(* Logix 5000 project; controller SX_V040001_C001 vendor 1 type 14 code 77 rev 16.22; software revision 16.04; part 7 of 35 *)
(* tags used below, declared in another part *)
   ALARM_BITS : INT[10];
   ALL_KINDS : INT[90];
   average_current : DINT;
   DRIVE : INT[32];
   DRIVE_INTERVAL : INT[8];
   EMPTYING : INT[18];
   FP_ALARM_EXIST : BOOL;
   G_AInput : DINT[8];
   G_DInput : DINT[3];
   G_DOutput : DINT[3];
   loading : INT[19];
   m_alarm_exist : BOOL;
   m_alarm_horn : BOOL;
   m_notstop : BOOL;
   METERING : INT[44];
   PARAMETER : INT[501];
   pointer_dump_current : DINT;
   RECIPE_GENERAL : INT[405];
   T_MET12_END : TIMER;
   T_MET13_END : TIMER;
   T_MET14_END : TIMER;
   T_MET_VALVE_13 : TIMER;
   T_MET_VALVE_14 : TIMER;
   TEMP : INT[14];
(* MainProgram, continued *)

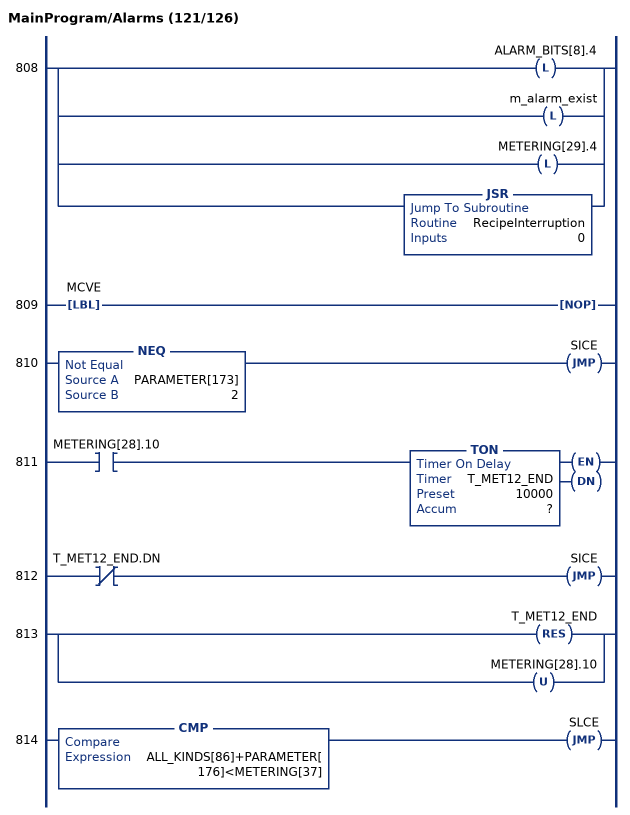
   [picture p142: MainProgram/Alarms rungs 808-814]
   808: [OTL(ALARM_BITS[8].4) ,OTL(m_alarm_exist) ,OTL(METERING[29].4) ,JSR(RecipeInterruption,0) ];
   809: LBL(MCVE)NOP();
   810: NEQ(PARAMETER[173],2)JMP(SICE);
   811: XIC(METERING[28].10)TON(T_MET12_END,?,?);
   812: XIO(T_MET12_END.DN)JMP(SICE);
   813: [RES(T_MET12_END) ,OTU(METERING[28].10) ];
   814: CMP(ALL_KINDS[86]+PARAMETER[176]<METERING[37])JMP(SLCE);
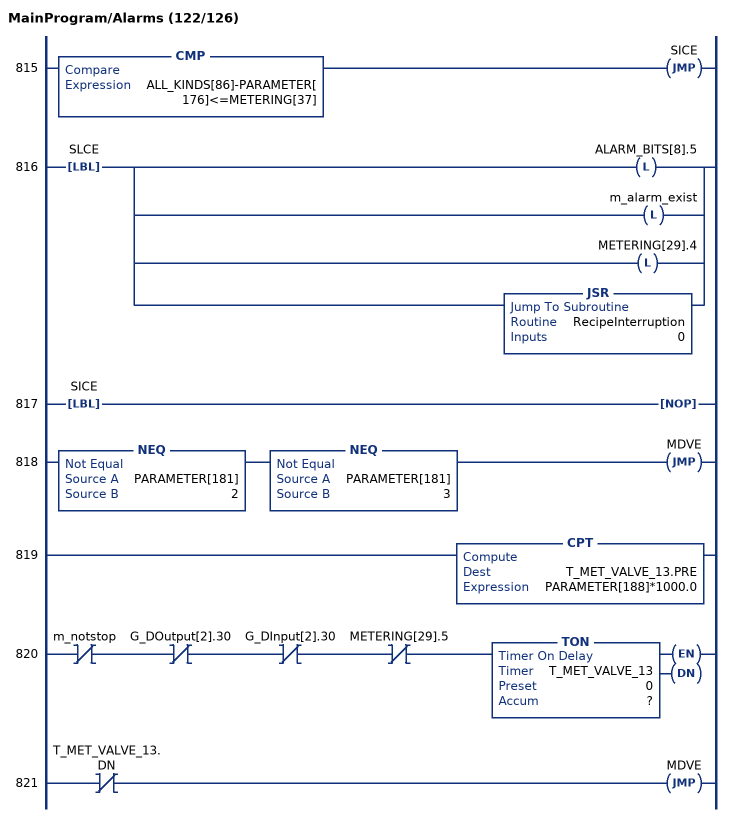
   815: CMP(ALL_KINDS[86]-PARAMETER[176]<=METERING[37])JMP(SICE);
   816: LBL(SLCE)[OTL(ALARM_BITS[8].5) ,OTL(m_alarm_exist) ,OTL(METERING[29].4) ,JSR(RecipeInterruption,0) ];
   817: LBL(SICE)NOP();
   818: NEQ(PARAMETER[181],2)NEQ(PARAMETER[181],3)JMP(MDVE);
   819: CPT(T_MET_VALVE_13.PRE,PARAMETER[188]*1000.0);
   820: XIO(m_notstop)XIO(G_DOutput[2].30)XIO(G_DInput[2].30)XIO(METERING[29].5)TON(T_MET_VALVE_13,?,?);
   821: XIO(T_MET_VALVE_13.DN)JMP(MDVE);
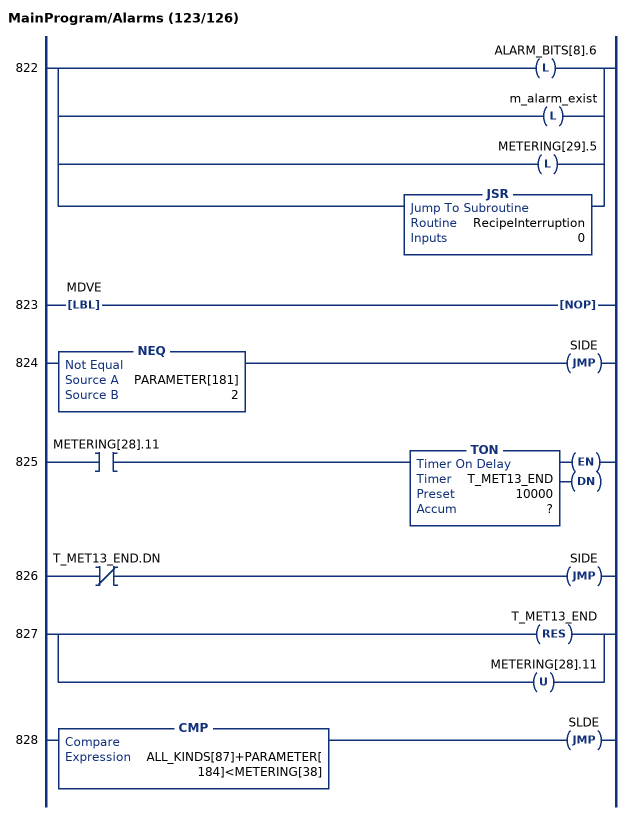
   822: [OTL(ALARM_BITS[8].6) ,OTL(m_alarm_exist) ,OTL(METERING[29].5) ,JSR(RecipeInterruption,0) ];
   823: LBL(MDVE)NOP();
   824: NEQ(PARAMETER[181],2)JMP(SIDE);
   825: XIC(METERING[28].11)TON(T_MET13_END,?,?);
   826: XIO(T_MET13_END.DN)JMP(SIDE);
   827: [RES(T_MET13_END) ,OTU(METERING[28].11) ];
   828: CMP(ALL_KINDS[87]+PARAMETER[184]<METERING[38])JMP(SLDE);
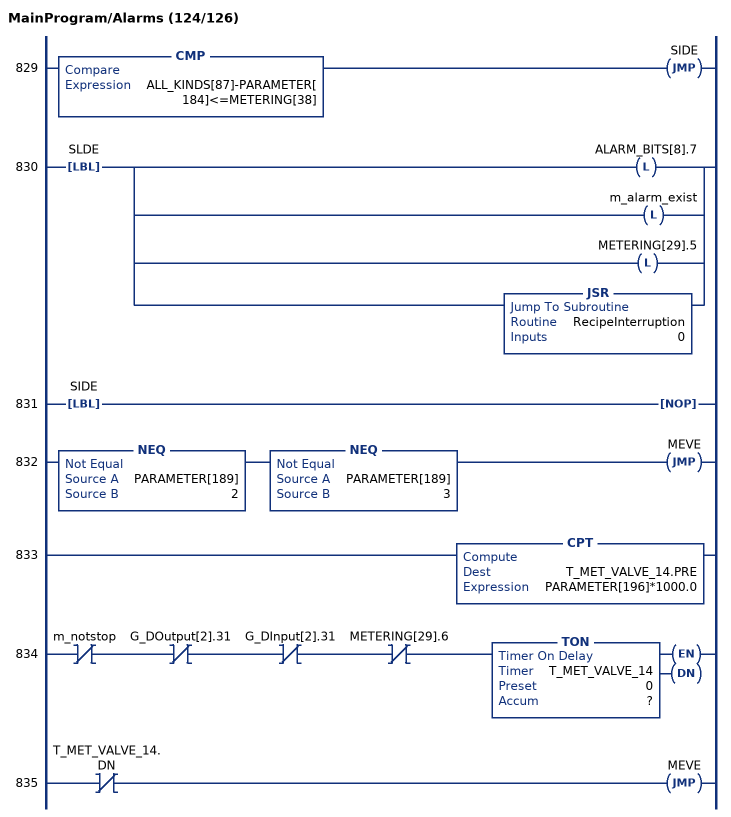
   829: CMP(ALL_KINDS[87]-PARAMETER[184]<=METERING[38])JMP(SIDE);
   830: LBL(SLDE)[OTL(ALARM_BITS[8].7) ,OTL(m_alarm_exist) ,OTL(METERING[29].5) ,JSR(RecipeInterruption,0) ];
   831: LBL(SIDE)NOP();
   832: NEQ(PARAMETER[189],2)NEQ(PARAMETER[189],3)JMP(MEVE);
   833: CPT(T_MET_VALVE_14.PRE,PARAMETER[196]*1000.0);
   834: XIO(m_notstop)XIO(G_DOutput[2].31)XIO(G_DInput[2].31)XIO(METERING[29].6)TON(T_MET_VALVE_14,?,?);
   835: XIO(T_MET_VALVE_14.DN)JMP(MEVE);
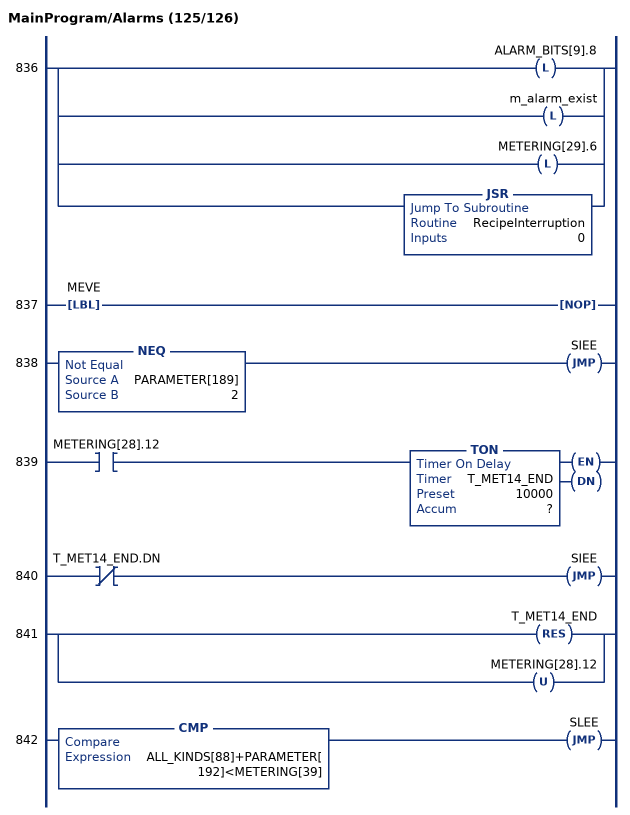
   836: [OTL(ALARM_BITS[9].8) ,OTL(m_alarm_exist) ,OTL(METERING[29].6) ,JSR(RecipeInterruption,0) ];
   837: LBL(MEVE)NOP();
   838: NEQ(PARAMETER[189],2)JMP(SIEE);
   839: XIC(METERING[28].12)TON(T_MET14_END,?,?);
   840: XIO(T_MET14_END.DN)JMP(SIEE);
   841: [RES(T_MET14_END) ,OTU(METERING[28].12) ];
   842: CMP(ALL_KINDS[88]+PARAMETER[192]<METERING[39])JMP(SLEE);
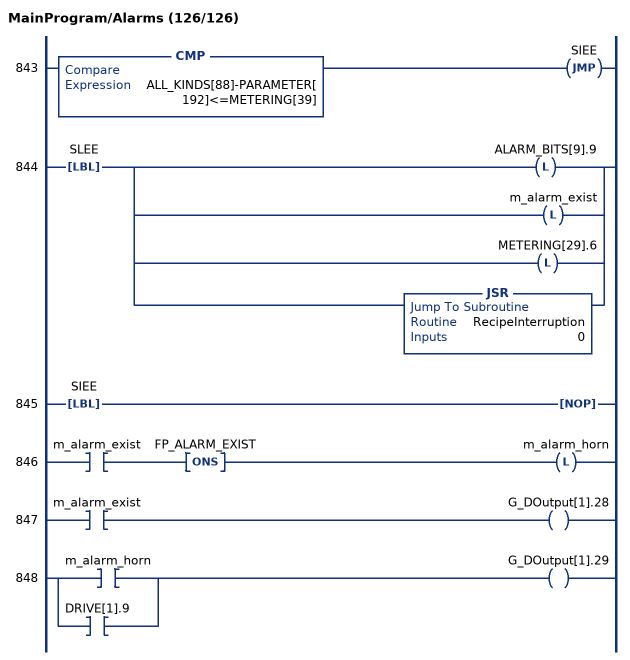
   843: CMP(ALL_KINDS[88]-PARAMETER[192]<=METERING[39])JMP(SIEE);
   844: LBL(SLEE)[OTL(ALARM_BITS[9].9) ,OTL(m_alarm_exist) ,OTL(METERING[29].6) ,JSR(RecipeInterruption,0) ];
   845: LBL(SIEE)NOP();
   846: XIC(m_alarm_exist)ONS(FP_ALARM_EXIST)OTL(m_alarm_horn);
   847: XIC(m_alarm_exist)OTE(G_DOutput[1].28);
   848: [XIC(m_alarm_horn) ,XIC(DRIVE[1].9) ]OTE(G_DOutput[1].29);
END_ROUTINE

ROUTINE AnalogInput   (* ladder *)
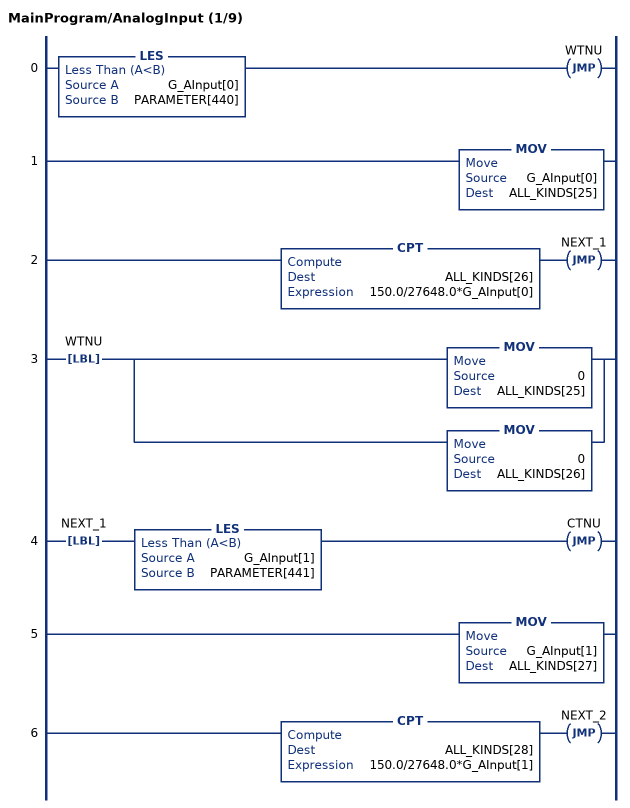
   0: LES(G_AInput[0],PARAMETER[440])JMP(WTNU);
   1: MOV(G_AInput[0],ALL_KINDS[25]);
   2: CPT(ALL_KINDS[26],150.0/27648.0*G_AInput[0])JMP(NEXT_1);
   3: LBL(WTNU)[MOV(0,ALL_KINDS[25]) ,MOV(0,ALL_KINDS[26]) ];
   4: LBL(NEXT_1)LES(G_AInput[1],PARAMETER[441])JMP(CTNU);
   5: MOV(G_AInput[1],ALL_KINDS[27]);
   6: CPT(ALL_KINDS[28],150.0/27648.0*G_AInput[1])JMP(NEXT_2);
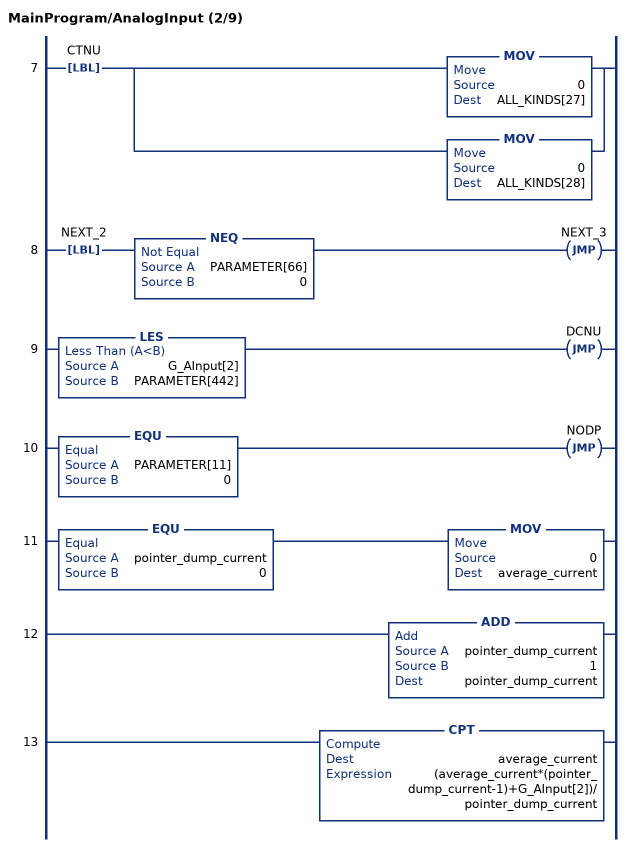
   7: LBL(CTNU)[MOV(0,ALL_KINDS[27]) ,MOV(0,ALL_KINDS[28]) ];
   8: LBL(NEXT_2)NEQ(PARAMETER[66],0)JMP(NEXT_3);
   9: LES(G_AInput[2],PARAMETER[442])JMP(DCNU);
   10: EQU(PARAMETER[11],0)JMP(NODP);
   11: EQU(pointer_dump_current,0)MOV(0,average_current);
   12: ADD(pointer_dump_current,1,pointer_dump_current);
   13: CPT(average_current,(average_current*(pointer_dump_current-1)+G_AInput[2])/pointer_dump_current);
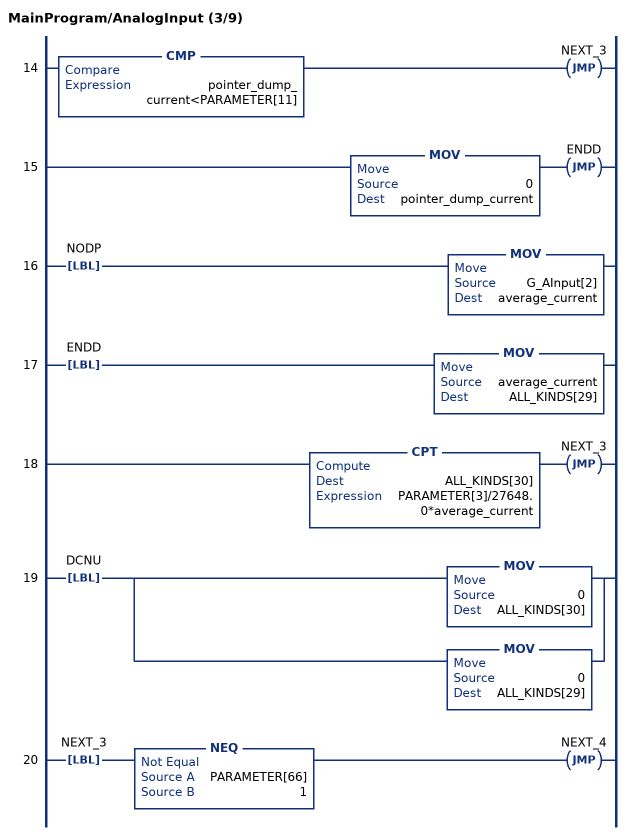
   14: CMP(pointer_dump_current<PARAMETER[11])JMP(NEXT_3);
   15: MOV(0,pointer_dump_current)JMP(ENDD);
   16: LBL(NODP)MOV(G_AInput[2],average_current);
   17: LBL(ENDD)MOV(average_current,ALL_KINDS[29]);
   18: CPT(ALL_KINDS[30],PARAMETER[3]/27648.0*average_current)JMP(NEXT_3);
   19: LBL(DCNU)[MOV(0,ALL_KINDS[30]) ,MOV(0,ALL_KINDS[29]) ];
   20: LBL(NEXT_3)NEQ(PARAMETER[66],1)JMP(NEXT_4);
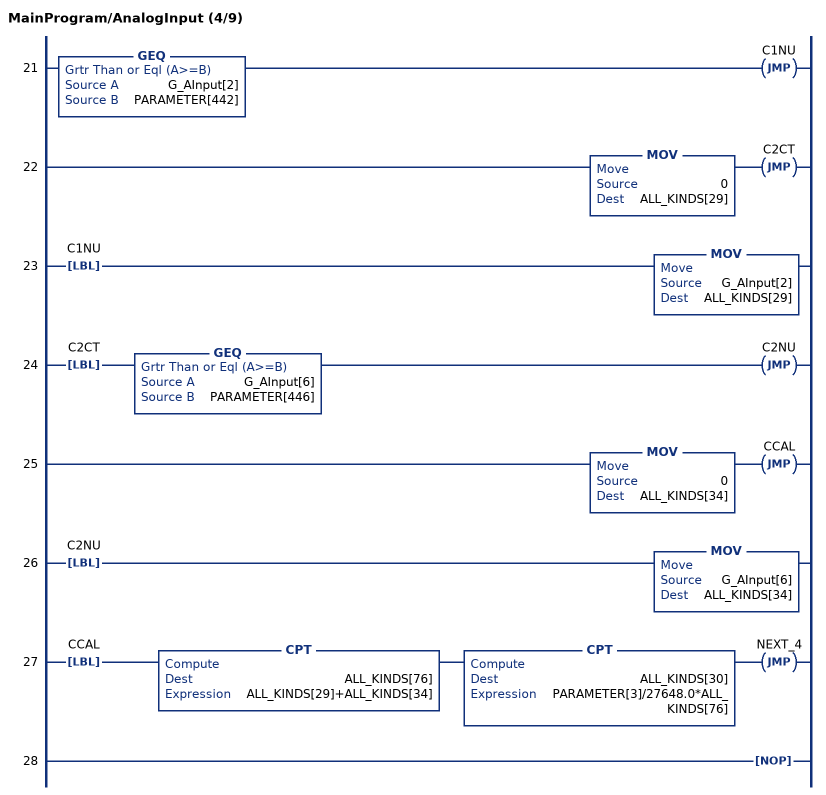
   21: GEQ(G_AInput[2],PARAMETER[442])JMP(C1NU);
   22: MOV(0,ALL_KINDS[29])JMP(C2CT);
   23: LBL(C1NU)MOV(G_AInput[2],ALL_KINDS[29]);
   24: LBL(C2CT)GEQ(G_AInput[6],PARAMETER[446])JMP(C2NU);
   25: MOV(0,ALL_KINDS[34])JMP(CCAL);
   26: LBL(C2NU)MOV(G_AInput[6],ALL_KINDS[34]);
   27: LBL(CCAL)CPT(ALL_KINDS[76],ALL_KINDS[29]+ALL_KINDS[34])CPT(ALL_KINDS[30],PARAMETER[3]/27648.0*ALL_KINDS[76])JMP(NEXT_4);
   28: NOP();
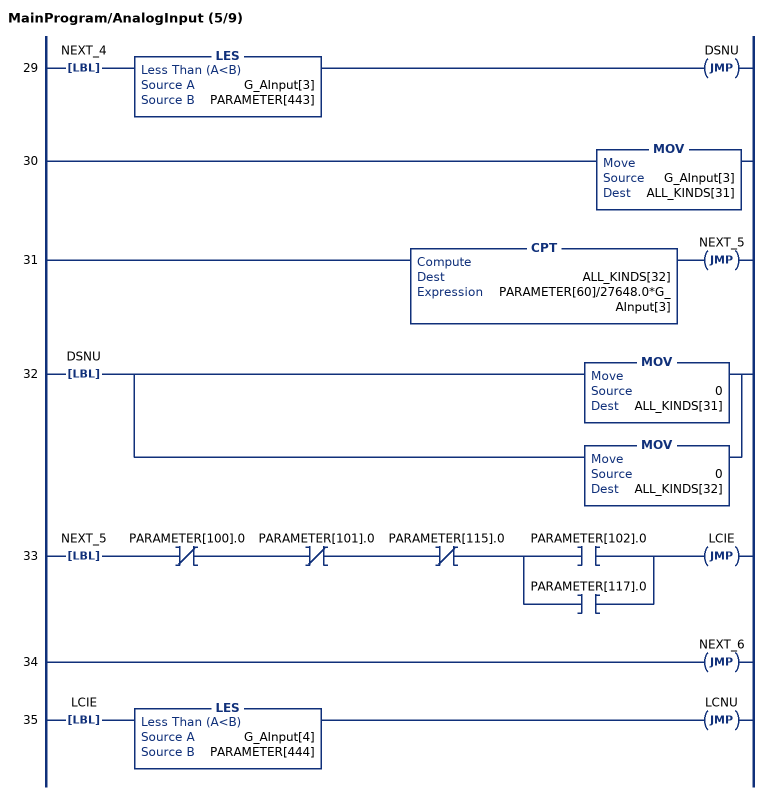
   29: LBL(NEXT_4)LES(G_AInput[3],PARAMETER[443])JMP(DSNU);
   30: MOV(G_AInput[3],ALL_KINDS[31]);
   31: CPT(ALL_KINDS[32],PARAMETER[60]/27648.0*G_AInput[3])JMP(NEXT_5);
   32: LBL(DSNU)[MOV(0,ALL_KINDS[31]) ,MOV(0,ALL_KINDS[32]) ];
   33: LBL(NEXT_5)XIO(PARAMETER[100].0)XIO(PARAMETER[101].0)XIO(PARAMETER[115].0)[XIC(PARAMETER[102].0) ,XIC(PARAMETER[117].0) ]JMP(LCIE);
   34: JMP(NEXT_6);
   35: LBL(LCIE)LES(G_AInput[4],PARAMETER[444])JMP(LCNU);
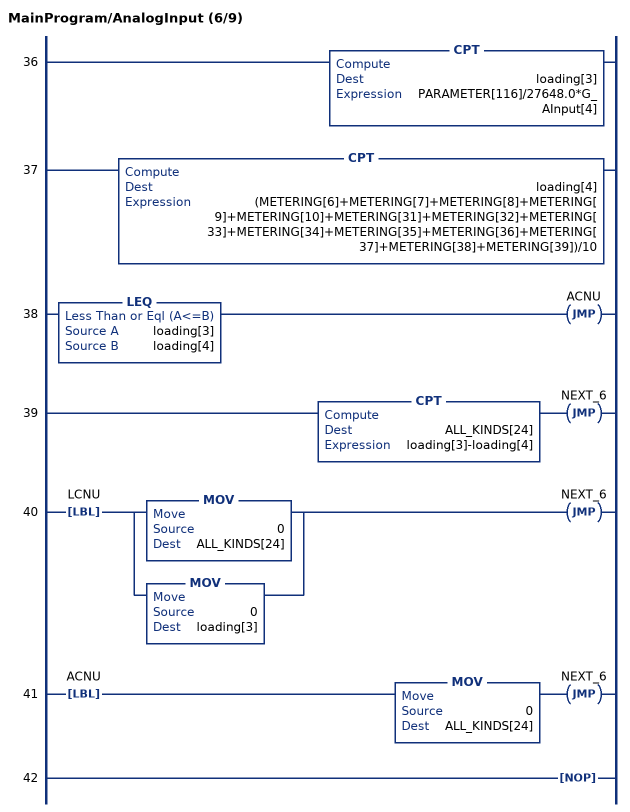
   36: CPT(loading[3],PARAMETER[116]/27648.0*G_AInput[4]);
   37: CPT(loading[4],(METERING[6]+METERING[7]+METERING[8]+METERING[9]+METERING[10]+METERING[31]+METERING[32]+METERING[33]+METERING[34]+METERING[35]+METERING[36]+METERING[37]+METERING[38]+METERING[39])/10);
   38: LEQ(loading[3],loading[4])JMP(ACNU);
   39: CPT(ALL_KINDS[24],loading[3]-loading[4])JMP(NEXT_6);
   40: LBL(LCNU)[MOV(0,ALL_KINDS[24]) ,MOV(0,loading[3]) ]JMP(NEXT_6);
   41: LBL(ACNU)MOV(0,ALL_KINDS[24])JMP(NEXT_6);
   42: NOP();
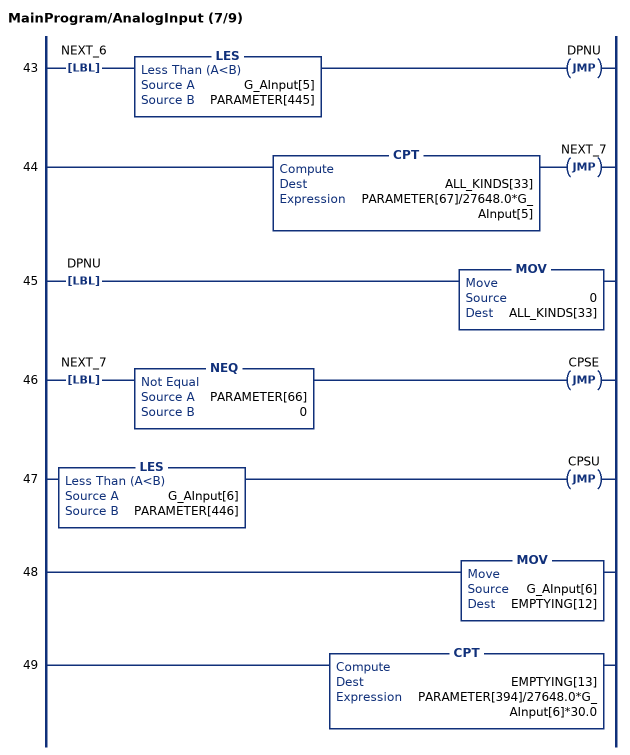
   43: LBL(NEXT_6)LES(G_AInput[5],PARAMETER[445])JMP(DPNU);
   44: CPT(ALL_KINDS[33],PARAMETER[67]/27648.0*G_AInput[5])JMP(NEXT_7);
   45: LBL(DPNU)MOV(0,ALL_KINDS[33]);
   46: LBL(NEXT_7)NEQ(PARAMETER[66],0)JMP(CPSE);
   47: LES(G_AInput[6],PARAMETER[446])JMP(CPSU);
   48: MOV(G_AInput[6],EMPTYING[12]);
   49: CPT(EMPTYING[13],PARAMETER[394]/27648.0*G_AInput[6]*30.0);
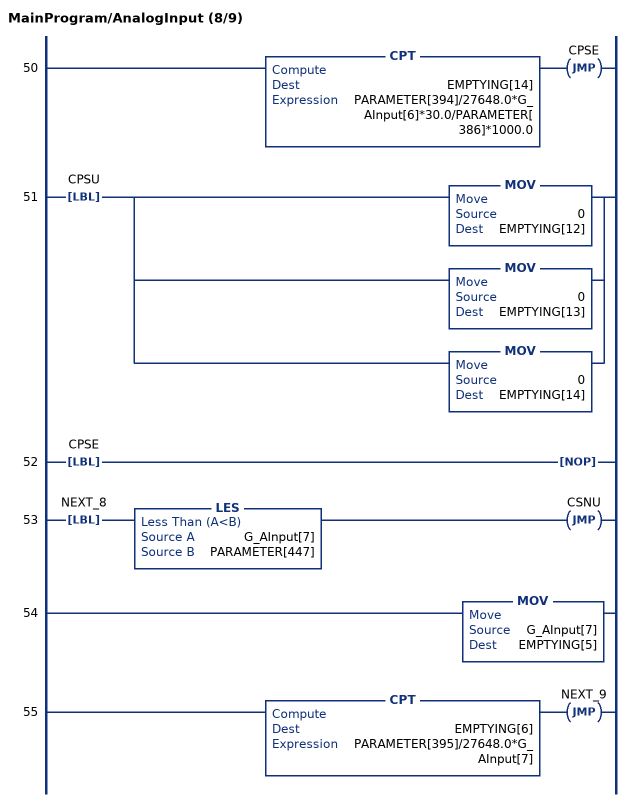
   50: CPT(EMPTYING[14],PARAMETER[394]/27648.0*G_AInput[6]*30.0/PARAMETER[386]*1000.0)JMP(CPSE);
   51: LBL(CPSU)[MOV(0,EMPTYING[12]) ,MOV(0,EMPTYING[13]) ,MOV(0,EMPTYING[14]) ];
   52: LBL(CPSE)NOP();
   53: LBL(NEXT_8)LES(G_AInput[7],PARAMETER[447])JMP(CSNU);
   54: MOV(G_AInput[7],EMPTYING[5]);
   55: CPT(EMPTYING[6],PARAMETER[395]/27648.0*G_AInput[7])JMP(NEXT_9);
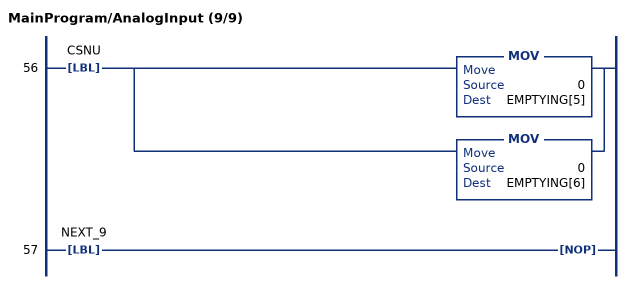
   56: LBL(CSNU)[MOV(0,EMPTYING[5]) ,MOV(0,EMPTYING[6]) ];
   57: LBL(NEXT_9)NOP();
END_ROUTINE

ROUTINE AnalyseRecipe   (* ladder *)
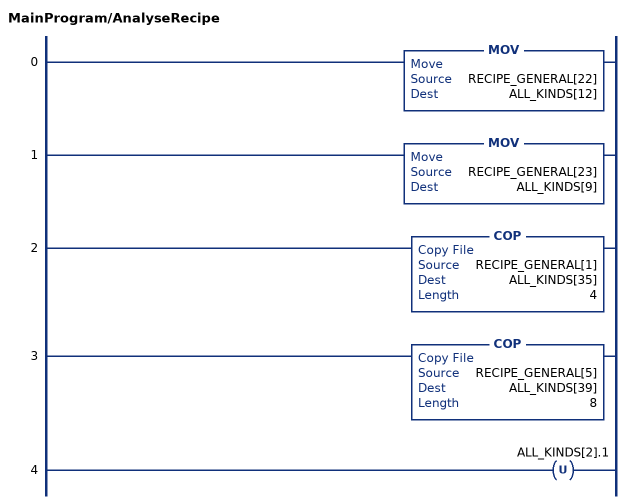
   0: MOV(RECIPE_GENERAL[22],ALL_KINDS[12]);
   1: MOV(RECIPE_GENERAL[23],ALL_KINDS[9]);
   2: COP(RECIPE_GENERAL[1],ALL_KINDS[35],4);
   3: COP(RECIPE_GENERAL[5],ALL_KINDS[39],8);
   4: OTU(ALL_KINDS[2].1);
END_ROUTINE

ROUTINE AnalyseRestart   (* ladder *)
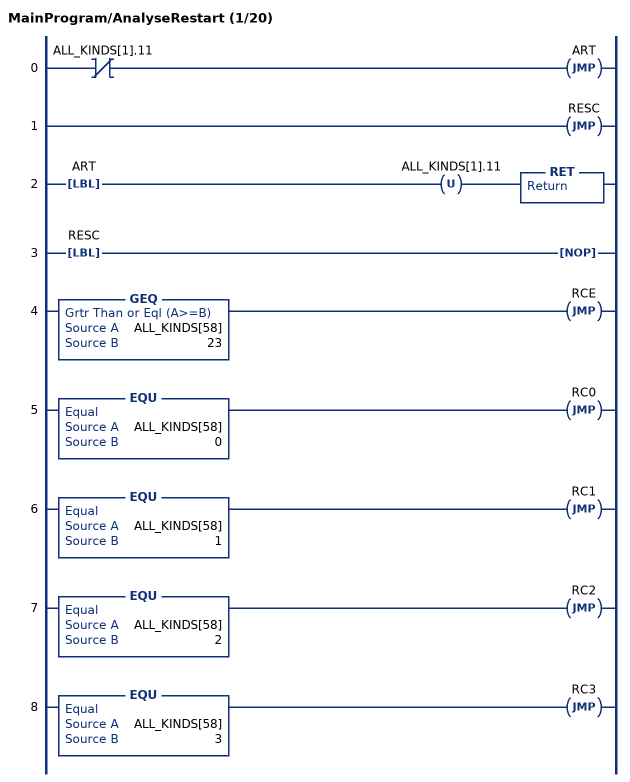
   0: XIO(ALL_KINDS[1].11)JMP(ART);
   1: JMP(RESC);
   2: LBL(ART)OTU(ALL_KINDS[1].11)RET();
   3: LBL(RESC)NOP();
   4: GEQ(ALL_KINDS[58],23)JMP(RCE);
   5: EQU(ALL_KINDS[58],0)JMP(RC0);
   6: EQU(ALL_KINDS[58],1)JMP(RC1);
   7: EQU(ALL_KINDS[58],2)JMP(RC2);
   8: EQU(ALL_KINDS[58],3)JMP(RC3);
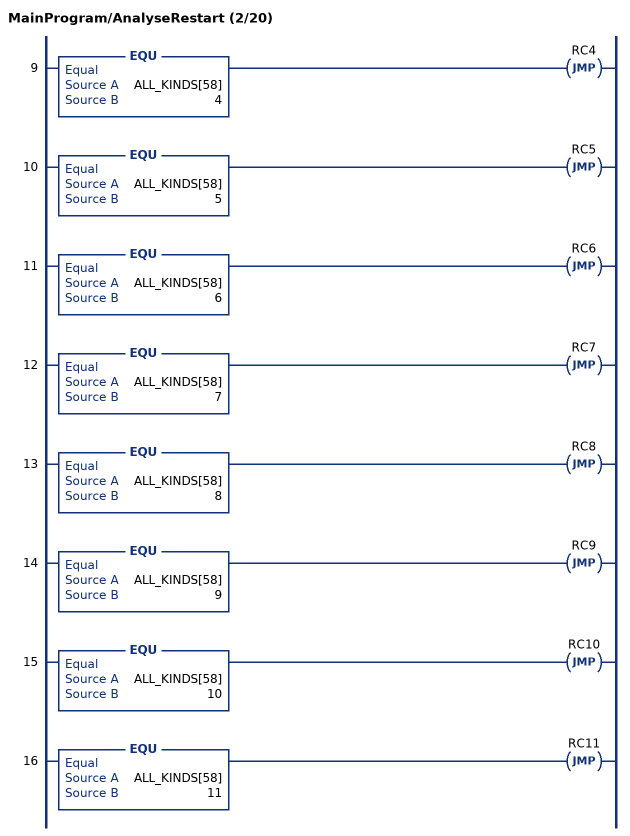
   9: EQU(ALL_KINDS[58],4)JMP(RC4);
   10: EQU(ALL_KINDS[58],5)JMP(RC5);
   11: EQU(ALL_KINDS[58],6)JMP(RC6);
   12: EQU(ALL_KINDS[58],7)JMP(RC7);
   13: EQU(ALL_KINDS[58],8)JMP(RC8);
   14: EQU(ALL_KINDS[58],9)JMP(RC9);
   15: EQU(ALL_KINDS[58],10)JMP(RC10);
   16: EQU(ALL_KINDS[58],11)JMP(RC11);
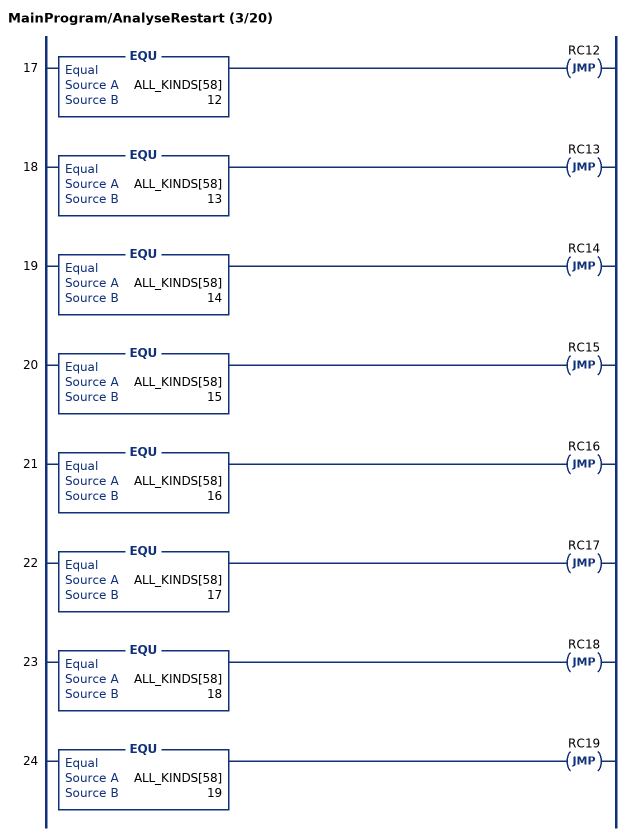
   17: EQU(ALL_KINDS[58],12)JMP(RC12);
   18: EQU(ALL_KINDS[58],13)JMP(RC13);
   19: EQU(ALL_KINDS[58],14)JMP(RC14);
   20: EQU(ALL_KINDS[58],15)JMP(RC15);
   21: EQU(ALL_KINDS[58],16)JMP(RC16);
   22: EQU(ALL_KINDS[58],17)JMP(RC17);
   23: EQU(ALL_KINDS[58],18)JMP(RC18);
   24: EQU(ALL_KINDS[58],19)JMP(RC19);
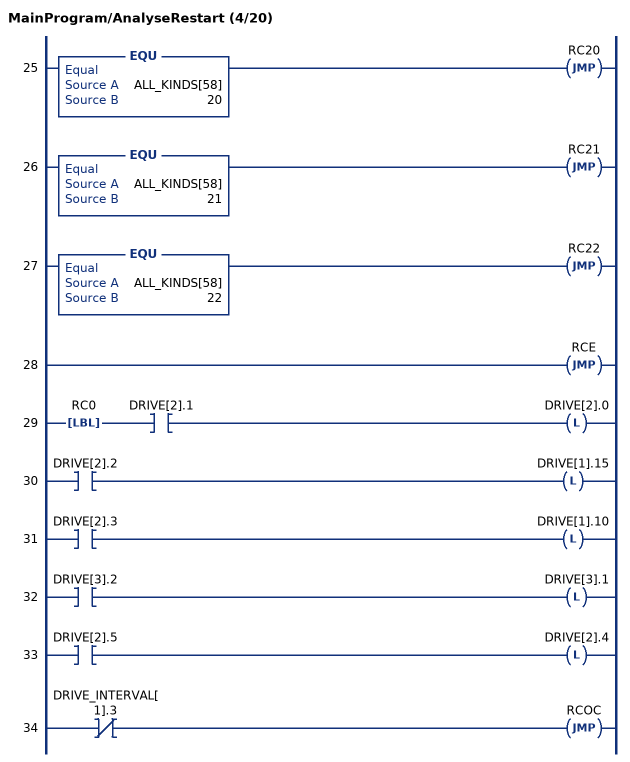
   25: EQU(ALL_KINDS[58],20)JMP(RC20);
   26: EQU(ALL_KINDS[58],21)JMP(RC21);
   27: EQU(ALL_KINDS[58],22)JMP(RC22);
   28: JMP(RCE);
   29: LBL(RC0)XIC(DRIVE[2].1)OTL(DRIVE[2].0);
   30: XIC(DRIVE[2].2)OTL(DRIVE[1].15);
   31: XIC(DRIVE[2].3)OTL(DRIVE[1].10);
   32: XIC(DRIVE[3].2)OTL(DRIVE[3].1);
   33: XIC(DRIVE[2].5)OTL(DRIVE[2].4);
   34: XIO(DRIVE_INTERVAL[1].3)JMP(RCOC);
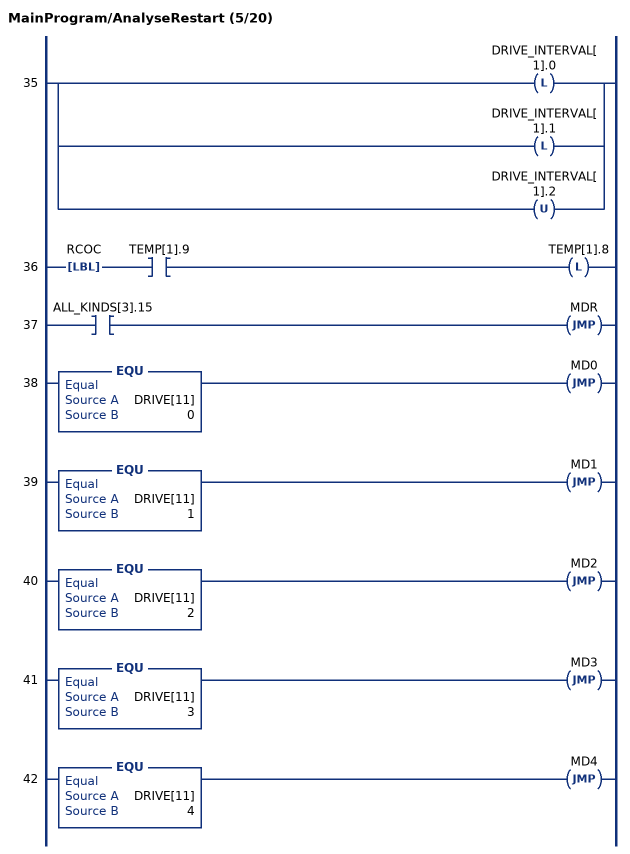
   35: [OTL(DRIVE_INTERVAL[1].0) ,OTL(DRIVE_INTERVAL[1].1) ,OTU(DRIVE_INTERVAL[1].2) ];
   36: LBL(RCOC)XIC(TEMP[1].9)OTL(TEMP[1].8);
   37: XIC(ALL_KINDS[3].15)JMP(MDR);
   38: EQU(DRIVE[11],0)JMP(MD0);
   39: EQU(DRIVE[11],1)JMP(MD1);
   40: EQU(DRIVE[11],2)JMP(MD2);
   41: EQU(DRIVE[11],3)JMP(MD3);
   42: EQU(DRIVE[11],4)JMP(MD4);
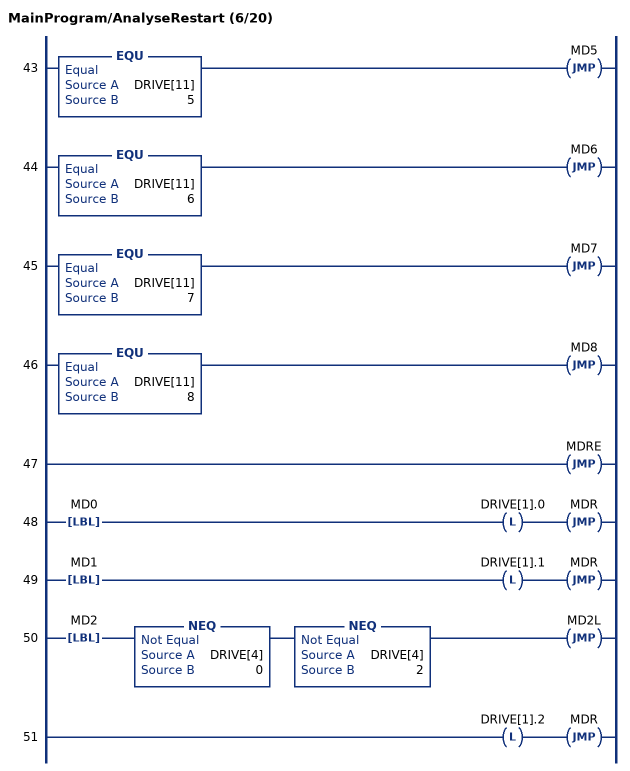
   43: EQU(DRIVE[11],5)JMP(MD5);
   44: EQU(DRIVE[11],6)JMP(MD6);
   45: EQU(DRIVE[11],7)JMP(MD7);
   46: EQU(DRIVE[11],8)JMP(MD8);
   47: JMP(MDRE);
   48: LBL(MD0)OTL(DRIVE[1].0)JMP(MDR);
   49: LBL(MD1)OTL(DRIVE[1].1)JMP(MDR);
   50: LBL(MD2)NEQ(DRIVE[4],0)NEQ(DRIVE[4],2)JMP(MD2L);
   51: OTL(DRIVE[1].2)JMP(MDR);
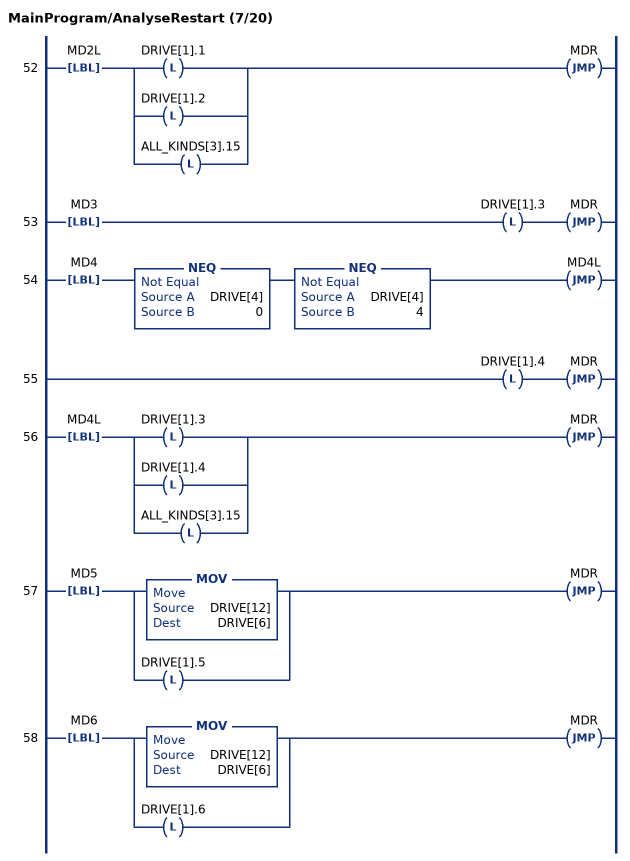
   52: LBL(MD2L)[OTL(DRIVE[1].1) ,OTL(DRIVE[1].2) ,OTL(ALL_KINDS[3].15) ]JMP(MDR);
   53: LBL(MD3)OTL(DRIVE[1].3)JMP(MDR);
   54: LBL(MD4)NEQ(DRIVE[4],0)NEQ(DRIVE[4],4)JMP(MD4L);
   55: OTL(DRIVE[1].4)JMP(MDR);
   56: LBL(MD4L)[OTL(DRIVE[1].3) ,OTL(DRIVE[1].4) ,OTL(ALL_KINDS[3].15) ]JMP(MDR);
   57: LBL(MD5)[MOV(DRIVE[12],DRIVE[6]) ,OTL(DRIVE[1].5) ]JMP(MDR);
   58: LBL(MD6)[MOV(DRIVE[12],DRIVE[6]) ,OTL(DRIVE[1].6) ]JMP(MDR);
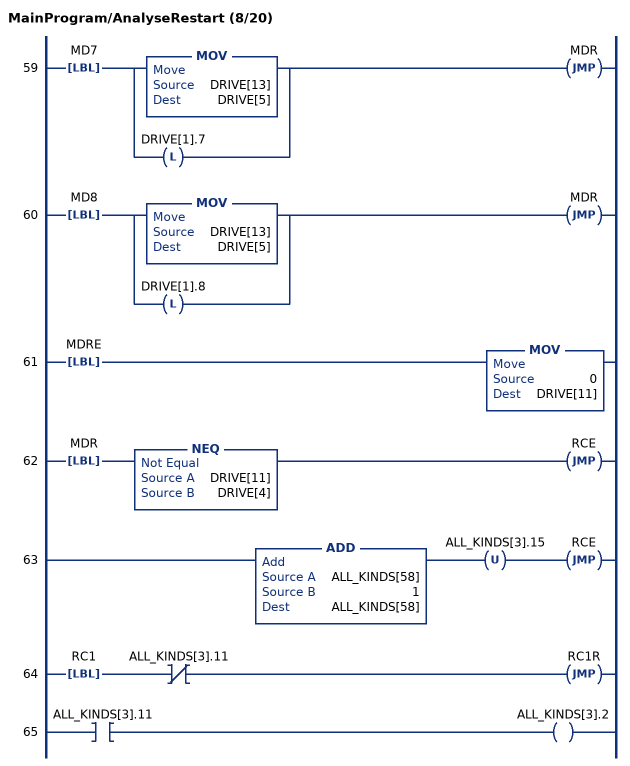
   59: LBL(MD7)[MOV(DRIVE[13],DRIVE[5]) ,OTL(DRIVE[1].7) ]JMP(MDR);
   60: LBL(MD8)[MOV(DRIVE[13],DRIVE[5]) ,OTL(DRIVE[1].8) ]JMP(MDR);
   61: LBL(MDRE)MOV(0,DRIVE[11]);
   62: LBL(MDR)NEQ(DRIVE[11],DRIVE[4])JMP(RCE);
   63: ADD(ALL_KINDS[58],1,ALL_KINDS[58])OTU(ALL_KINDS[3].15)JMP(RCE);
   64: LBL(RC1)XIO(ALL_KINDS[3].11)JMP(RC1R);
   65: XIC(ALL_KINDS[3].11)OTE(ALL_KINDS[3].2);
